LIN {X 0,Y 79.401,Z 461.557,A -85,B 0,C 180,E1 -30801.674,E2 -30801.674} C_VEL
LIN {X 0,Y 73.583,Z 474.091,A -85,B 0,C 180,E1 -30803.189,E2 -30803.189} C_VEL
LIN {X 0,Y 68.268,Z 483.249,A -85,B 0,C 180,E1 -30804.775,E2 -30804.775} C_VEL
LIN {X 0,Y 64.835,Z 488.082,A -85,B 0,C 180,E1 -30805.163,E2 -30805.163} C_VEL
LIN {X 0,Y 58.34,Z 495.556,A -85,B 0,C 180,E1 -30804.458,E2 -30804.458} C_VEL
LIN {X 0,Y 51.356,Z 502.55,A -85,B 0,C 180,E1 -30803.746,E2 -30803.746} C_VEL
LIN {X 0,Y 47.097,Z 506.573,A -85,B 0,C 180,E1 -30804.501,E2 -30804.501} C_VEL
LIN {X 0,Y 38.123,Z 514.34,A -85,B 0,C 180,E1 -30808.895,E2 -30808.895} C_VEL
LIN {X 0,Y 28.505,Z 521.316,A -85,B 0,C 180,E1 -30816.765,E2 -30816.765} C_VEL
LIN {X 0,Y 18.48,Z 527.736,A -85,B 0,C 180,E1 -30835.237,E2 -30835.237} C_VEL
LIN {X 0,Y 12.939,Z 531.979,A -85,B 0,C 180,E1 -30870.023,E2 -30870.023} C_VEL
LIN {X 0,Y 13.206,Z 534.216,A -85,B 0,C 180,E1 -30902.179,E2 -30902.179} C_VEL
LIN {X 0,Y 16.879,Z 535.973,A -85,B 0,C 180,E1 -30926.415,E2 -30926.415} C_VEL
LIN {X 0,Y 23.365,Z 537.518,A -85,B 0,C 180,E1 -30942.493,E2 -30942.493} C_VEL
LIN {X 0,Y 35.283,Z 538.711,A -85,B 0,C 180,E1 -30954.933,E2 -30954.933} C_VEL
LIN {X 0,Y 45.214,Z 538.684,A -85,B 0,C 180,E1 -30960,E2 -30960} C_VEL
LIN {X 0,Y 56.34,Z 537.642,A -85,B 0,C 180,E1 -30963.608,E2 -30963.608} C_VEL
LIN {X 0,Y 63.522,Z 536.408,A -85,B 0,C 180,E1 -30965.248,E2 -30965.248} C_VEL
LIN {X 0,Y 63.625,Z 536.421,A -85,B 0,C 180,E1 -30966.172,E2 -30966.172} C_VEL
LIN {X 0,Y 49.874,Z 538.62,A -85,B 0,C 180,E1 -30969.428,E2 -30969.428} C_VEL
LIN {X 0,Y 36.417,Z 539.218,A -85,B 0,C 180,E1 -30975.191,E2 -30975.191} C_VEL
LIN {X 0,Y 23.839,Z 538.327,A -85,B 0,C 180,E1 -30987.793,E2 -30987.793} C_VEL
LIN {X 0,Y 18.437,Z 537.3,A -85,B 0,C 180,E1 -31000.302,E2 -31000.302} C_VEL
LIN {X 0,Y 14.532,Z 535.846,A -85,B 0,C 180,E1 -31021.055,E2 -31021.055} C_VEL
LIN {X 0,Y 13.155,Z 533.966,A -85,B 0,C 180,E1 -31049.978,E2 -31049.978} C_VEL
LIN {X 0,Y 16.092,Z 530.169,A -85,B 0,C 180,E1 -31090.904,E2 -31090.904} C_VEL
LIN {X 0,Y 23.682,Z 525.198,A -85,B 0,C 180,E1 -31112.883,E2 -31112.883} C_VEL
LIN {X 0,Y 33.009,Z 518.935,A -85,B 0,C 180,E1 -31123.321,E2 -31123.321} C_VEL
LIN {X 0,Y 42.862,Z 511.034,A -85,B 0,C 180,E1 -31129.63,E2 -31129.63} C_VEL
LIN {X 0,Y 51.388,Z 503.009,A -85,B 0,C 180,E1 -31132.492,E2 -31132.492} C_VEL
LIN {X 0,Y 59.119,Z 494.242,A -85,B 0,C 180,E1 -31134.569,E2 -31134.569} C_VEL
LIN {X 0,Y 66.038,Z 484.796,A -85,B 0,C 180,E1 -31136.049,E2 -31136.049} C_VEL
LIN {X 0,Y 73,Z 473.113,A -85,B 0,C 180,E1 -31137.146,E2 -31137.146} C_VEL
LIN {X 0,Y 78.602,Z 460.858,A -85,B 0,C 180,E1 -31137.935,E2 -31137.935} C_VEL
LIN {X 0,Y 82.945,Z 447.956,A -85,B 0,C 180,E1 -31138.399,E2 -31138.399} C_VEL
LIN {X 0,Y 85.891,Z 434.744,A -85,B 0,C 180,E1 -31138.763,E2 -31138.763} C_VEL
LIN {X 0,Y 87.332,Z 423.644,A -85,B 0,C 180,E1 -31139.129,E2 -31139.129} C_VEL
LIN {X 0,Y 86.983,Z 420.627,A -85,B 0,C 180,E1 -31144.054,E2 -31144.054} C_VEL
LIN {X 0,Y 86.921,Z 421.064,A -85,B 0,C 180,E1 -31150.386,E2 -31150.386} C_VEL
LIN {X 0,Y 87.268,Z 423.672,A -85,B 0,C 180,E1 -31155.173,E2 -31155.173} C_VEL
LIN {X 0,Y 87.252,Z 424.212,A -85,B 0,C 180,E1 -31155.422,E2 -31155.422} C_VEL
LIN {X 0,Y 85.185,Z 437.926,A -85,B 0,C 180,E1 -31155.689,E2 -31155.689} C_VEL
LIN {X 0,Y 82.207,Z 449.864,A -85,B 0,C 180,E1 -31156.074,E2 -31156.074} C_VEL
LIN {X 0,Y 77.922,Z 461.85,A -85,B 0,C 180,E1 -31156.621,E2 -31156.621} C_VEL
LIN {X 0,Y 71.945,Z 474.376,A -85,B 0,C 180,E1 -31157.758,E2 -31157.758} C_VEL
LIN {X 0,Y 66.6,Z 483.321,A -85,B 0,C 180,E1 -31158.913,E2 -31158.913} C_VEL
LIN {X 0,Y 59.155,Z 493.554,A -85,B 0,C 180,E1 -31160.691,E2 -31160.691} C_VEL
LIN {X 0,Y 51.498,Z 502.227,A -85,B 0,C 180,E1 -31162.916,E2 -31162.916} C_VEL
LIN {X 0,Y 47.097,Z 506.573,A -85,B 0,C 180,E1 -31164.501,E2 -31164.501} C_VEL
LIN {X 0,Y 42.694,Z 510.443,A -85,B 0,C 180,E1 -31165.442,E2 -31165.442} C_VEL
LIN {X 0,Y 34.666,Z 516.248,A -85,B 0,C 180,E1 -31164.937,E2 -31164.937} C_VEL
LIN {X 0,Y 26.191,Z 521.416,A -85,B 0,C 180,E1 -31164.246,E2 -31164.246} C_VEL
LIN {X 0,Y 21.084,Z 524.289,A -85,B 0,C 180,E1 -31166.348,E2 -31166.348} C_VEL
LIN {X 0,Y 10.105,Z 529.899,A -85,B 0,C 180,E1 -31185.972,E2 -31185.972} C_VEL
LIN {X 0,Y 5.908,Z 533.693,A -85,B 0,C 180,E1 -31266.559,E2 -31266.559} C_VEL
LIN {X 0,Y 14.202,Z 536.437,A -85,B 0,C 180,E1 -31311.925,E2 -31311.925} C_VEL
LIN {X 0,Y 21.089,Z 537.739,A -85,B 0,C 180,E1 -31319.999,E2 -31319.999} C_VEL
LIN {X 0,Y 28.198,Z 538.586,A -85,B 0,C 180,E1 -31324.34,E2 -31324.34} C_VEL
LIN {X 0,Y 28.291,Z 538.632,A -85,B 0,C 180,E1 -31326.357,E2 -31326.357} C_VEL
LIN {X 0,Y 21.465,Z 537.959,A -85,B 0,C 180,E1 -31330.749,E2 -31330.749} C_VEL
LIN {X 0,Y 8.992,Z 535.366,A -85,B 0,C 180,E1 -31358.54,E2 -31358.54} C_VEL
LIN {X 0,Y 6.043,Z 533.444,A -85,B 0,C 180,E1 -31409.952,E2 -31409.952} C_VEL
LIN {X 0,Y 11.676,Z 529.558,A -85,B 0,C 180,E1 -31474.477,E2 -31474.477} C_VEL
LIN {X 0,Y 21.392,Z 524.493,A -85,B 0,C 180,E1 -31490.185,E2 -31490.185} C_VEL
LIN {X 0,Y 31.705,Z 518.116,A -85,B 0,C 180,E1 -31495.814,E2 -31495.814} C_VEL
LIN {X 0,Y 42.165,Z 510.035,A -85,B 0,C 180,E1 -31499.334,E2 -31499.334} C_VEL
LIN {X 0,Y 50.949,Z 501.871,A -85,B 0,C 180,E1 -31500.527,E2 -31500.527} C_VEL
LIN {X 0,Y 58.874,Z 492.934,A -85,B 0,C 180,E1 -31501.525,E2 -31501.525} C_VEL
LIN {X 0,Y 65.932,Z 483.281,A -85,B 0,C 180,E1 -31502.237,E2 -31502.237} C_VEL
LIN {X 0,Y 72.111,Z 472.907,A -85,B 0,C 180,E1 -31502.705,E2 -31502.705} C_VEL
LIN {X 0,Y 77.858,Z 460.491,A -85,B 0,C 180,E1 -31503.096,E2 -31503.096} C_VEL
LIN {X 0,Y 82.249,Z 447.53,A -85,B 0,C 180,E1 -31503.295,E2 -31503.295} C_VEL
LIN {X 0,Y 85.141,Z 434.726,A -85,B 0,C 180,E1 -31503.492,E2 -31503.492} C_VEL
LIN {X 0,Y 86.058,Z 428.337,A -85,B 0,C 180,E1 -31503.621,E2 -31503.621} C_VEL
LIN {X 0,Y 86.045,Z 427.772,A -85,B 0,C 180,E1 -31504.685,E2 -31504.685} C_VEL
LIN {X 0,Y 85.993,Z 428.004,A -85,B 0,C 180,E1 -31509.408,E2 -31509.408} C_VEL
LIN {X 0,Y 85.997,Z 428.7,A -85,B 0,C 180,E1 -31510.746,E2 -31510.746} C_VEL
LIN {X 0,Y 83.669,Z 441.72,A -85,B 0,C 180,E1 -31511.032,E2 -31511.032} C_VEL
LIN {X 0,Y 80.299,Z 453.536,A -85,B 0,C 180,E1 -31511.146,E2 -31511.146} C_VEL
LIN {X 0,Y 75.326,Z 466.116,A -85,B 0,C 180,E1 -31511.598,E2 -31511.598} C_VEL
LIN {X 0,Y 69.246,Z 477.708,A -85,B 0,C 180,E1 -31512.372,E2 -31512.372} C_VEL
LIN {X 0,Y 62.326,Z 488.151,A -85,B 0,C 180,E1 -31513.22,E2 -31513.22} C_VEL
LIN {X 0,Y 54.411,Z 497.877,A -85,B 0,C 180,E1 -31514.39,E2 -31514.39} C_VEL
LIN {X 0,Y 45.584,Z 506.764,A -85,B 0,C 180,E1 -31515.94,E2 -31515.94} C_VEL
LIN {X 0,Y 35.228,Z 515.238,A -85,B 0,C 180,E1 -31518.655,E2 -31518.655} C_VEL
LIN {X 0,Y 24.896,Z 522.097,A -85,B 0,C 180,E1 -31523.476,E2 -31523.476} C_VEL
LIN {X 0,Y 21.084,Z 524.289,A -85,B 0,C 180,E1 -31526.348,E2 -31526.348} C_VEL
LIN {X 0,Y 20.073,Z 526.056,A -85,B 0,C 180,E1 -31527.262,E2 -31527.262} C_VEL
LIN {X 0,Y 20.073,Z 600,A -85,B 0,C 180,E1 -31527.262,E2 -31527.262} C_VEL
LIN {X 0,Y 20.073,Z 600,A -85,B 0,C 180,E1 -31527.262,E2 -31527.262}

QRS_NEXT_CUT()

QRS_NEXT()
QRS_HOME()

END
